FUNCTION_BLOCK Test_NotificationHandlerOnlyAddedOnce EXTENDS T_UnitTestBase
VAR
    Source   : T_Notification;
    Handler  : T_NotificationHandler;
    IsRaised : BOOL;
	Assertion : T_Assertion;
END_VAR

{attribute 'analysis' := '-33'} // inhibit unused variable warning
METHOD RunTest
VAR_OUTPUT
    TestCompleted : BOOL;
    TestFailed    : BOOL;
END_VAR
Handler.FB_init(bInitRetains := FALSE,
                bInCopyCode  := FALSE);

Source
	.ClearNotificationHandlers()
	.AddNotificationHandler(Handler)
	.AddNotificationHandler(Handler);

Source.Raise();
IsRaised := Handler.IsRaised();

TestFailed S= NOT Assertion.AssertEquals_BOOL(Source    := TestName,
                             Expected     := TRUE,
                            Actual       := IsRaised,
                            VariableName := 'IsRaised');

IsRaised := Handler.IsRaised();

TestFailed S= NOT Assertion.AssertEquals_BOOL(Source    := TestName,
                             Expected     := FALSE,
                            Actual       := IsRaised,
                            VariableName := 'IsRaised');

TestCompleted := TRUE;
END_METHOD

END_FUNCTION_BLOCK

(* stored: Version 1.1.0.1, ProductVersion 3.1.4024.12
   POU Test_NotificationHandlerOnlyAddedOnce: Id {d822493b-b417-457e-b68d-ce48b3adc9d5}, SpecialFunc None
   Method RunTest: Id {e4801cbe-a69b-4c40-b3f3-077fc4956321} *)
